TYPE PRINTF_DATA : ARRAY [1..11]  OF STRING(LOG_SIZE);
END_TYPE

(* stored: Version 1.1.0.1, ProductVersion 3.1.4024.4
   DUT PRINTF_DATA: Id {919aefa2-d142-41b2-af4d-fe7b35dd4d67} *)
